// Mitsubishi GX Works2 project: test   PLC: FX3U/FX3UC

// task Task_01 (event TRUE, interval 0, priority 31): POU_01

PROGRAM POU_01
VAR
  TON_win : TON;  (* 贏的畫面顯示延時 *)
  TON_loss : TON;  (* 輸掉的畫面顯示延時 *)
  R_TRIG_timer : R_TRIG;  (* 計時器上緣 *)
  R_TRIG_finger : R_TRIG;  (* 按鈕上綠 *)
  R_TRIG_flag : R_TRIG;  (* 按鈕上綠 *)
  R_TRIG_reset : R_TRIG;  (* 按鈕上綠 *)
  TON_timer : TON;  (* 遊戲計時器 *)
  temp_b : BOOL;
  temp_c : BOOL;
  wstep : INT;  (* 步數 *)
  map : map;  (* 地圖物件 *)
  blank : INT;  (* 按下的格數 *)
  win : INT;  (* 贏的條件 *)
  rand_seed : INT;  (* 亂數種子 *)
  vector : ARRAY [0..80] OF INT;  (* 容器 *)
  isum : INT;  (* 容器標號 *)
  temp_a : BOOL;  (* 檢測該格是否已被放入容器 *)
  cr : ARRAY [0..1] OF INT;
  ar : ARRAY [0..11] OF INT;
  click_mode : BOOL;  (* 點擊模式 旗子或手指 *)
  ii : INT;
  ij : INT;
  ia : INT;
  ib : INT;
  ix : INT;
  iy : INT;
  iz : INT;
END_VAR
(*
更新日記:

v1.0
初版完成

v1.1
HMI 圖示更新
更新看門狗
BUG修復
新增按鈕顯示
*)
*
(*初始化 或 按下重置按鈕*)
IF M8002 THEN
	WDT(TRUE);
	wstep := 0;
END_IF;
D8000 := 1000;

(*
M
開始遊戲 M90
重置遊戲 M91
踩地雷 M92
棋子 M93
贏顯示 M94
輸顯示 M95
切換開關顯示
	手指 M96
	旗子 M97
地圖按鈕 M0 ~ M80

D
地圖顯示 D0 ~ D80
	顯示已按下 10
	顯示周圍地雷數 11 ~ 18
	地雷 20
	棋子 21
秒數 D90
插旗數 D91

*)

(*重置按鈕*)
R_TRIG_reset(_CLK := M91);

(*計時模組*)
TON_timer(IN := (wstep >= 20) AND (wstep < 30 ) AND 
(NOT TON_timer.Q) , PT := T#1s); (*不斷計時，條件為處於遊戲狀態*)
R_TRIG_timer(_CLK := TON_timer.Q); (*計時上緣*)
IF R_TRIG_timer.Q THEN (*計時器+1*)
	D90 := D90 + 1;
END_IF;

(*插旗與手指切換*)
IF (wstep <> 0) THEN
	R_TRIG_finger(_CLK := M92);
	R_TRIG_flag(_CLK := M93);
	IF R_TRIG_finger.Q THEN
		M96 := TRUE;
		M97 := FALSE;
	END_IF;
	IF R_TRIG_flag.Q THEN
		M96 := FALSE;
		M97 := TRUE;		
	END_IF;
END_IF;

CASE wstep OF
	0: (*初始狀態*)
	FOR ii := 0 TO 80 BY 1 DO
		Z0 := ii;
		D0Z0 := 0;
		M0Z0 := FALSE;
		vector[ii] := 100;
	END_FOR;	
	
	(*產生亂數種子*)
	rand_seed := rand_seed + 1;
	IF rand_seed > 30000 THEN
		rand_seed := 0;
	END_IF;
	
	(*按下開始按鈕*)
	IF M90 OR R_TRIG_reset.Q THEN
		D90 := 0;
		D91 := 10;
		M92 := TRUE;
		map(generate := TRUE, bomb_rand := rand_seed);
		win := 0;
		wstep := 20;
	END_IF;
	
	20: (*遊戲中*)
	IF R_TRIG_reset.Q THEN
		wstep := 0;
	END_IF;
	
	temp_c := FALSE;
	FOR ii := 0 TO 80 BY 1 DO
		Z1 := ii;
		
		(*贏的條件*)
		IF (map.map[ii] <> 20) AND ( (D0Z1 >= 10) AND (D0Z1 <= 19) ) THEN (*若為 按下 或 插旗 則+1*)
			win := win + 1;
		END_IF;
		IF win = 71 THEN (*9顆地雷全被找到*)
			wstep := 40;
		END_IF; 		
		IF ii = 80 THEN (*歸零*)
			win := 0;
		END_IF;
		
		IF M0Z1 AND NOT temp_b THEN (*當按下格子*) (*1*)
			temp_b := TRUE;
			IF M96 AND (D0Z1 = 0 OR D0Z1 = 21) THEN (*處於手指觸發模式*) (*確保該格非被翻開*) (*2*)
				IF D0Z1 = 21 THEN (*若該格有棋子，則移除棋子並不執行任何動作*) (*3*)
					D0Z1 := 0;
					D91 := D91 + 1;
				ELSIF map.map[Z1] = 20 THEN (*踩到地雷*)
						D0Z1 := map.map[Z1];
						wstep := 30;
				ELSIF around_bomb(map.map, Z1) = 0 THEN (*踩到空白塊*)
					blank := Z1;
					wstep := 21;				
				ELSE (*周圍有地雷*) 
					D0Z1 := 10 + around_bomb(map.map, Z1);
				END_IF;	 (*3*)
			ELSIF M97 THEN (*插棋模式*) (*2*)
				(*交替顯示*)
				IF D0Z1 = 21 THEN
					D0Z1 := 0; 
					D91 := D91 + 1;
				ELSIF D0Z1 = 0 THEN
					D0Z1 := 21;
					D91 := D91 - 1;	
				END_IF;
			END_IF; (*2*)
		END_IF; (*1*)
		
		(*上緣觸發*)
		IF M0Z1 THEN
			temp_c := TRUE;
		END_IF;		
		
	END_FOR;
	temp_b := temp_c; (*確保所有按鈕都已放開*)
	
	21: (*翻牌*)
	isum := 0;
	vector[isum] := blank; (*創建容器 放置待翻開的格子*) 
	isum := isum + 1; (*容器標號*)
	FOR ix := 0 TO isum BY 1 DO (*1*) (*處理容器內的值 直到結束*)	
		ar := around(vector[ix]); (*周圍8格*)
		FOR iy := 8 TO 11 BY 1 DO (*2*) (*讀取周圍4格*)
			IF (ar[iy] <> 100) THEN (*3*)(*無越界*)
				IF (around_bomb(map.map, ar[iy]) = 0) THEN (*4*) (*周圍無炸彈*)		
					temp_a := FALSE;
					FOR iz := 0 TO isum BY 1 DO (*5*) (*檢查是否已有被加入容器*)
						IF vector[iz] = ar[iy] THEN (*6*)
							temp_a := TRUE;
						END_IF; (*6*)
					END_FOR; (*5*)
							
					IF NOT temp_a THEN (*5*) (*若無則放入容器*)
						vector[isum] := ar[iy];
						isum := isum + 1;
					END_IF; (*5*)	
				ELSE (*4*)
					Z4 := ar[iy];
					D0Z4 := 10 + around_bomb(map.map, Z4); (*打開旁邊的格子，並顯示周圍炸彈數*)
				END_IF; (*4*)		
			END_IF; (*3*)
		END_FOR; (*2*)					
	END_FOR; (*1*)	
	
	(*翻開所有容器內的牌*)
	FOR ix := 0 TO isum BY 1 DO (*1*) 
		Z4 := vector[ix];
		IF D0Z4 <> 20 THEN (*不翻開棋子*)
			D0Z4 := 10; (*標示為已按下*)
		END_IF;
	END_FOR; (*1*)
	wstep := 20;	

	30:
	TON_loss(IN := NOT TON_loss.Q, PT := T#1s);
	IF TON_loss.Q THEN
		wstep := 31;
	END_IF;
	
	31: (*翻開所有牌*)
	FOR ii := 0 TO 80 BY 1 DO
		Z2 := ii;
		IF map.map[ii] <> 20 THEN
			D0Z2 := 10 + around_bomb(map.map, Z2); (*顯示周圍炸彈數*)
		ELSE
			D0Z2 := 20;
		END_IF;
	END_FOR;	
	
	TON_loss(IN := NOT TON_loss.Q, PT := T#1s);
	IF TON_loss.Q THEN
		wstep := 32;
	END_IF;
	
	32: (* "你輸了" 顯示*)
	M95 := TRUE;
	TON_loss(IN := NOT TON_loss.Q, PT := T#2s);
	IF TON_loss.Q THEN
		M95 := FALSE;
		wstep := 0;
	END_IF;
	
	40: (* "你贏了" 顯示"*)
	M94 := TRUE;
	TON_win(IN := NOT TON_win.Q, PT := T#3s);
	IF TON_win.Q THEN
		M94 := FALSE;
		wstep := 0;
	END_IF;
		
END_CASE;
END_PROGRAM

FUNCTION_BLOCK map
VAR_INPUT
  generate : BOOL;
  bomb_rand : INT;  (* 種子輸入 *)
END_VAR
VAR
  times : ARRAY [0..6] OF INT;  (* 當前時間 *)
  temp_a : INT;  (* 時間 與 種子輸入 的亂數子 *)
  map : ARRAY [0..80] OF INT;  (* 地圖陣列 *)
  bomb : ARRAY [0..8] OF INT;  (* 炸彈9顆 *)
END_VAR
VAR CONSTANT
  bomb_tag : INT := 20;
END_VAR
VAR
  ii : INT;
  ij : INT;
END_VAR
IF generate THEN
	(*初使化地圖 為10*)
	FOR ii := 0 TO 80 BY 1 DO
		map[ii] := 10;
	END_FOR;
	
	(*產生地雷*)
	TRD(TRUE, times);
	WXOR(TRUE, bomb_rand * times[4], times[5] * times[6], temp_a); (*亂數種子*)
	bomb := rand(temp_a);
	FOR ii := 0 TO 8 BY 1 DO
		map[ (bomb[ii] MOD 80) ] := bomb_tag; (*放置炸彈*)
	END_FOR;

END_IF;
END_FUNCTION_BLOCK

FUNCTION around_bomb
VAR_INPUT
  map_in : ARRAY [0..80] OF INT;
  scan : INT;
END_VAR
VAR CONSTANT
  bomb_tag : INT := 20;
END_VAR
VAR
  result : INT;
  ii : INT;
  ar : ARRAY [0..11] OF INT;
  ar_block : INT;
END_VAR
ar := around(scan); (*讀取周圍八格*)

result := 0;
FOR ii := 0 TO 7 BY 1 DO
	IF (ar[ii] <> 100) AND (map_in[ ar[ii] ] = 20) THEN (*非炸彈且無越界*)
		result := result + 1;
	END_IF;
END_FOR;

around_bomb := result;
END_FUNCTION

FUNCTION cr_num_converter
VAR_INPUT
  column : INT;
  row : INT;
END_VAR
cr_num_converter := (column * 9) + row; (*行列轉數字*)
END_FUNCTION

FUNCTION num_cr_converter
VAR_INPUT
  num : INT;
END_VAR
VAR
  column : INT;
  row : INT;
  ii : INT;
  temp_a : BOOL;  (* 如果找到最接近的最大值則關閉計算 *)
END_VAR
temp_a := FALSE; (*暫存器*)
FOR ii := 1 TO 9 BY 1 DO
	IF ( (ii * 9) > num) AND (NOT temp_a) THEN (*找到最接近的數 設為行-1 暫存器關閉*)
		column := ii - 1;
		temp_a := TRUE;
	END_IF;
END_FOR;

row := num - (column * 9); (*由行反推出列*)

num_cr_converter[0] := column;
num_cr_converter[1] := row;
END_FUNCTION

FUNCTION around
VAR_INPUT
  scan : INT;
END_VAR
VAR
  result : ARRAY [0..11] OF INT;
  ii : INT;
  ij : INT;
  im : INT;
  cr : ARRAY [0..1] OF INT;
END_VAR
cr  := num_cr_converter(scan); (*數字轉行數*)

im := 0;

FOR ii := -1 TO 1 BY 1 DO (*行*)
	FOR ij := -1 TO 1 BY 1 DO (*列*)
		IF NOT ( 
			(*檢查有無超越邊界*)
			((cr[0] + ii) > 8) OR 
			((cr[0] + ii) < 0) OR 
			((cr[1] + ij) > 8) OR 
			((cr[1] + ij) < 0) 
			) THEN
			result[im] := cr_num_converter(cr[0] + ii, cr[1] + ij);
		ELSE (*若越界則設為100*)
			result[im] := 100;
		END_IF;
		
		(*自身格不算*)
		IF NOT (ii = 0 AND ij = 0) THEN
			im := im + 1;
		END_IF;
		
	END_FOR;
END_FOR; 

(*陣列後方為周圍四格 (不含角塊)*)
result[8] := result[1];
result[9] := result[3];
result[10] := result[4];
result[11] := result[6];

around := result;
END_FUNCTION

FUNCTION rand
VAR_INPUT
  seed : INT;
END_VAR
VAR
  result : ARRAY [0..8] OF INT;
  ii : INT;
  ij : INT;
END_VAR
result[0] :=  ABS( (seed + 1093) ) MOD 15031; (*第一亂數*)

FOR ii := 0 TO 7 BY 1 DO
	result[ii + 1] := ABS( (result[ii] + 1853) ) MOD 15061; (*線性同餘法*)
END_FOR;
rand := result;
END_FUNCTION
